// TIA Portal V20 export
FUNCTION_BLOCK "EventsPFE"   // FB95, LAD
// stored: MemoryReserve 100, Namespace Unit1.Em11, SetENOAutomatically false
   VAR
      data : Array[1..100] of LReal;
   END_VAR
BEGIN

REGION Network 1: Call PFE Events
   // Add the required PFE Events
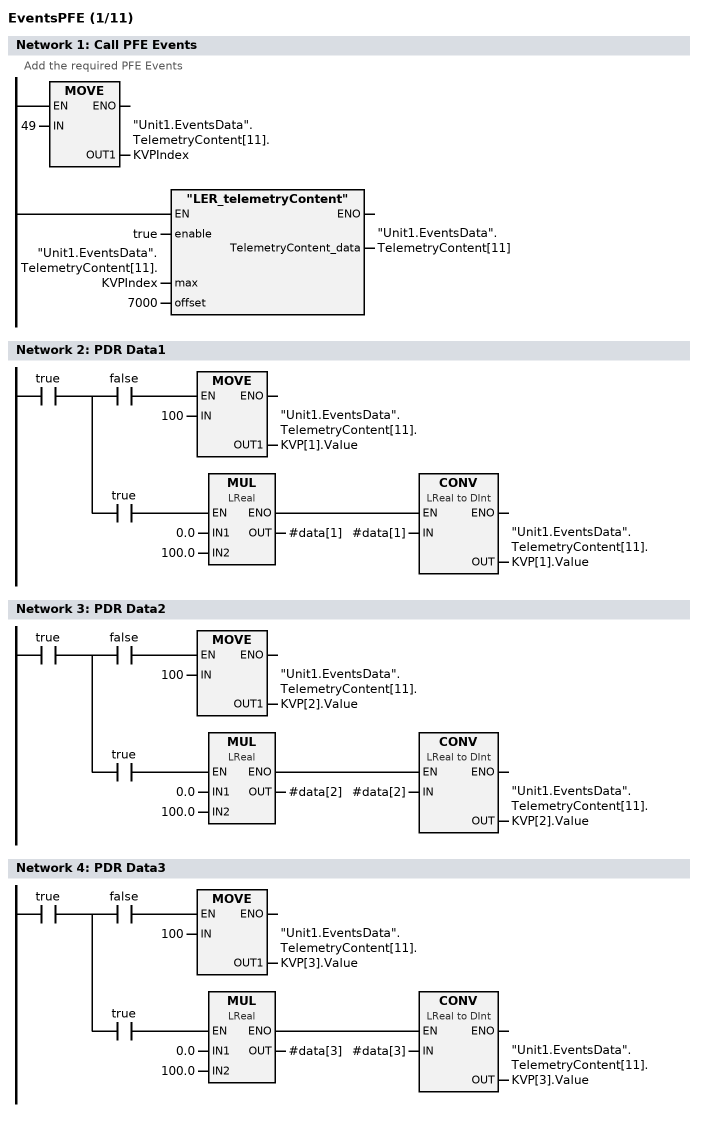
   RUNG wire#powerrail
      Move(in := 49, out1 => "Unit1.EventsData".TelemetryContent[11].KVPIndex)
   END_RUNG
   RUNG wire#powerrail
      "LER_telemetryContent"(enable := true, max := "Unit1.EventsData".TelemetryContent[11].KVPIndex, offset := 7000, TelemetryContent_data => "Unit1.EventsData".TelemetryContent[11])
   END_RUNG
   // the same network as SCL:
   "Unit1.EventsData".TelemetryContent[11].KVPIndex := 49;
   "LER_telemetryContent"(enable := true,
                          max := "Unit1.EventsData".TelemetryContent[11].KVPIndex,
                          offset := 7000,
                          TelemetryContent_data => "Unit1.EventsData".TelemetryContent[11]);
END_REGION

REGION Network 2: PDR Data1
   RUNG wire#powerrail
      Contact( true )
      wire#w1
      Contact( false )
      Move(in := 100, out1 => "Unit1.EventsData".TelemetryContent[11].KVP[1].Value)
   END_RUNG
   RUNG wire#w1
      Contact( true )
      { S7_Templates := "SrcType := LReal" } Mul(in1 := 0.0, in2 := 100.0, out => #data[1])
      { S7_Templates := "[SrcType := LReal, DestType := DInt]" } Convert(in := #data[1], out => "Unit1.EventsData".TelemetryContent[11].KVP[1].Value)
   END_RUNG
   // the same network as SCL:
   IF true AND false THEN "Unit1.EventsData".TelemetryContent[11].KVP[1].Value := 100; END_IF;
   IF true AND true THEN
       #data[1] := 0.0 * 100.0;
       "Unit1.EventsData".TelemetryContent[11].KVP[1].Value := LREAL_TO_DINT(#data[1]);
   END_IF;
END_REGION

REGION Network 3: PDR Data2
   RUNG wire#powerrail
      Contact( true )
      wire#w1
      Contact( false )
      Move(in := 100, out1 => "Unit1.EventsData".TelemetryContent[11].KVP[2].Value)
   END_RUNG
   RUNG wire#w1
      Contact( true )
      { S7_Templates := "SrcType := LReal" } Mul(in1 := 0.0, in2 := 100.0, out => #data[2])
      { S7_Templates := "[SrcType := LReal, DestType := DInt]" } Convert(in := #data[2], out => "Unit1.EventsData".TelemetryContent[11].KVP[2].Value)
   END_RUNG
   // the same network as SCL:
   IF true AND false THEN "Unit1.EventsData".TelemetryContent[11].KVP[2].Value := 100; END_IF;
   IF true AND true THEN
       #data[2] := 0.0 * 100.0;
       "Unit1.EventsData".TelemetryContent[11].KVP[2].Value := LREAL_TO_DINT(#data[2]);
   END_IF;
END_REGION

REGION Network 4: PDR Data3
   RUNG wire#powerrail
      Contact( true )
      wire#w1
      Contact( false )
      Move(in := 100, out1 => "Unit1.EventsData".TelemetryContent[11].KVP[3].Value)
   END_RUNG
   RUNG wire#w1
      Contact( true )
      { S7_Templates := "SrcType := LReal" } Mul(in1 := 0.0, in2 := 100.0, out => #data[3])
      { S7_Templates := "[SrcType := LReal, DestType := DInt]" } Convert(in := #data[3], out => "Unit1.EventsData".TelemetryContent[11].KVP[3].Value)
   END_RUNG
   // the same network as SCL:
   IF true AND false THEN "Unit1.EventsData".TelemetryContent[11].KVP[3].Value := 100; END_IF;
   IF true AND true THEN
       #data[3] := 0.0 * 100.0;
       "Unit1.EventsData".TelemetryContent[11].KVP[3].Value := LREAL_TO_DINT(#data[3]);
   END_IF;
END_REGION

REGION Network 5: PDR Data4
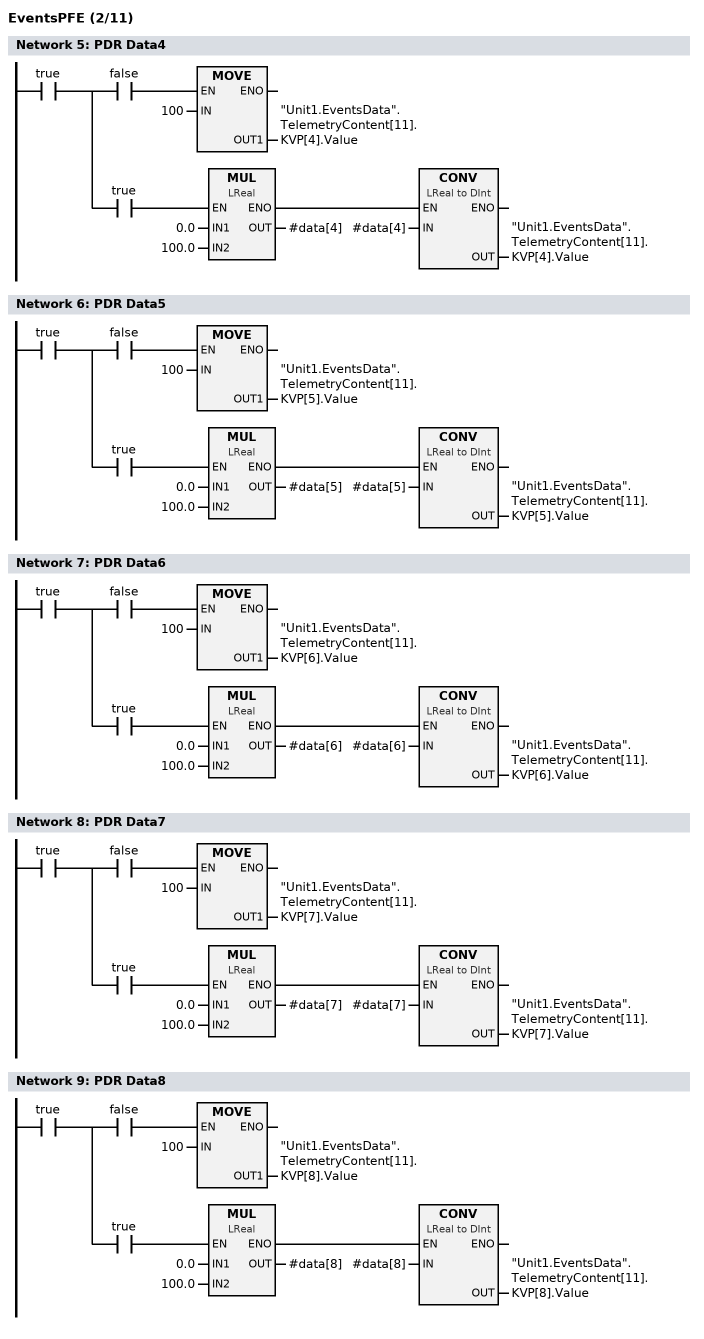
   RUNG wire#powerrail
      Contact( true )
      wire#w1
      Contact( false )
      Move(in := 100, out1 => "Unit1.EventsData".TelemetryContent[11].KVP[4].Value)
   END_RUNG
   RUNG wire#w1
      Contact( true )
      { S7_Templates := "SrcType := LReal" } Mul(in1 := 0.0, in2 := 100.0, out => #data[4])
      { S7_Templates := "[SrcType := LReal, DestType := DInt]" } Convert(in := #data[4], out => "Unit1.EventsData".TelemetryContent[11].KVP[4].Value)
   END_RUNG
   // the same network as SCL:
   IF true AND false THEN "Unit1.EventsData".TelemetryContent[11].KVP[4].Value := 100; END_IF;
   IF true AND true THEN
       #data[4] := 0.0 * 100.0;
       "Unit1.EventsData".TelemetryContent[11].KVP[4].Value := LREAL_TO_DINT(#data[4]);
   END_IF;
END_REGION

REGION Network 6: PDR Data5
   RUNG wire#powerrail
      Contact( true )
      wire#w1
      Contact( false )
      Move(in := 100, out1 => "Unit1.EventsData".TelemetryContent[11].KVP[5].Value)
   END_RUNG
   RUNG wire#w1
      Contact( true )
      { S7_Templates := "SrcType := LReal" } Mul(in1 := 0.0, in2 := 100.0, out => #data[5])
      { S7_Templates := "[SrcType := LReal, DestType := DInt]" } Convert(in := #data[5], out => "Unit1.EventsData".TelemetryContent[11].KVP[5].Value)
   END_RUNG
   // the same network as SCL:
   IF true AND false THEN "Unit1.EventsData".TelemetryContent[11].KVP[5].Value := 100; END_IF;
   IF true AND true THEN
       #data[5] := 0.0 * 100.0;
       "Unit1.EventsData".TelemetryContent[11].KVP[5].Value := LREAL_TO_DINT(#data[5]);
   END_IF;
END_REGION

REGION Network 7: PDR Data6
   RUNG wire#powerrail
      Contact( true )
      wire#w1
      Contact( false )
      Move(in := 100, out1 => "Unit1.EventsData".TelemetryContent[11].KVP[6].Value)
   END_RUNG
   RUNG wire#w1
      Contact( true )
      { S7_Templates := "SrcType := LReal" } Mul(in1 := 0.0, in2 := 100.0, out => #data[6])
      { S7_Templates := "[SrcType := LReal, DestType := DInt]" } Convert(in := #data[6], out => "Unit1.EventsData".TelemetryContent[11].KVP[6].Value)
   END_RUNG
   // the same network as SCL:
   IF true AND false THEN "Unit1.EventsData".TelemetryContent[11].KVP[6].Value := 100; END_IF;
   IF true AND true THEN
       #data[6] := 0.0 * 100.0;
       "Unit1.EventsData".TelemetryContent[11].KVP[6].Value := LREAL_TO_DINT(#data[6]);
   END_IF;
END_REGION

REGION Network 8: PDR Data7
   RUNG wire#powerrail
      Contact( true )
      wire#w1
      Contact( false )
      Move(in := 100, out1 => "Unit1.EventsData".TelemetryContent[11].KVP[7].Value)
   END_RUNG
   RUNG wire#w1
      Contact( true )
      { S7_Templates := "SrcType := LReal" } Mul(in1 := 0.0, in2 := 100.0, out => #data[7])
      { S7_Templates := "[SrcType := LReal, DestType := DInt]" } Convert(in := #data[7], out => "Unit1.EventsData".TelemetryContent[11].KVP[7].Value)
   END_RUNG
   // the same network as SCL:
   IF true AND false THEN "Unit1.EventsData".TelemetryContent[11].KVP[7].Value := 100; END_IF;
   IF true AND true THEN
       #data[7] := 0.0 * 100.0;
       "Unit1.EventsData".TelemetryContent[11].KVP[7].Value := LREAL_TO_DINT(#data[7]);
   END_IF;
END_REGION

REGION Network 9: PDR Data8
   RUNG wire#powerrail
      Contact( true )
      wire#w1
      Contact( false )
      Move(in := 100, out1 => "Unit1.EventsData".TelemetryContent[11].KVP[8].Value)
   END_RUNG
   RUNG wire#w1
      Contact( true )
      { S7_Templates := "SrcType := LReal" } Mul(in1 := 0.0, in2 := 100.0, out => #data[8])
      { S7_Templates := "[SrcType := LReal, DestType := DInt]" } Convert(in := #data[8], out => "Unit1.EventsData".TelemetryContent[11].KVP[8].Value)
   END_RUNG
   // the same network as SCL:
   IF true AND false THEN "Unit1.EventsData".TelemetryContent[11].KVP[8].Value := 100; END_IF;
   IF true AND true THEN
       #data[8] := 0.0 * 100.0;
       "Unit1.EventsData".TelemetryContent[11].KVP[8].Value := LREAL_TO_DINT(#data[8]);
   END_IF;
END_REGION

REGION Network 10: PDR Data9
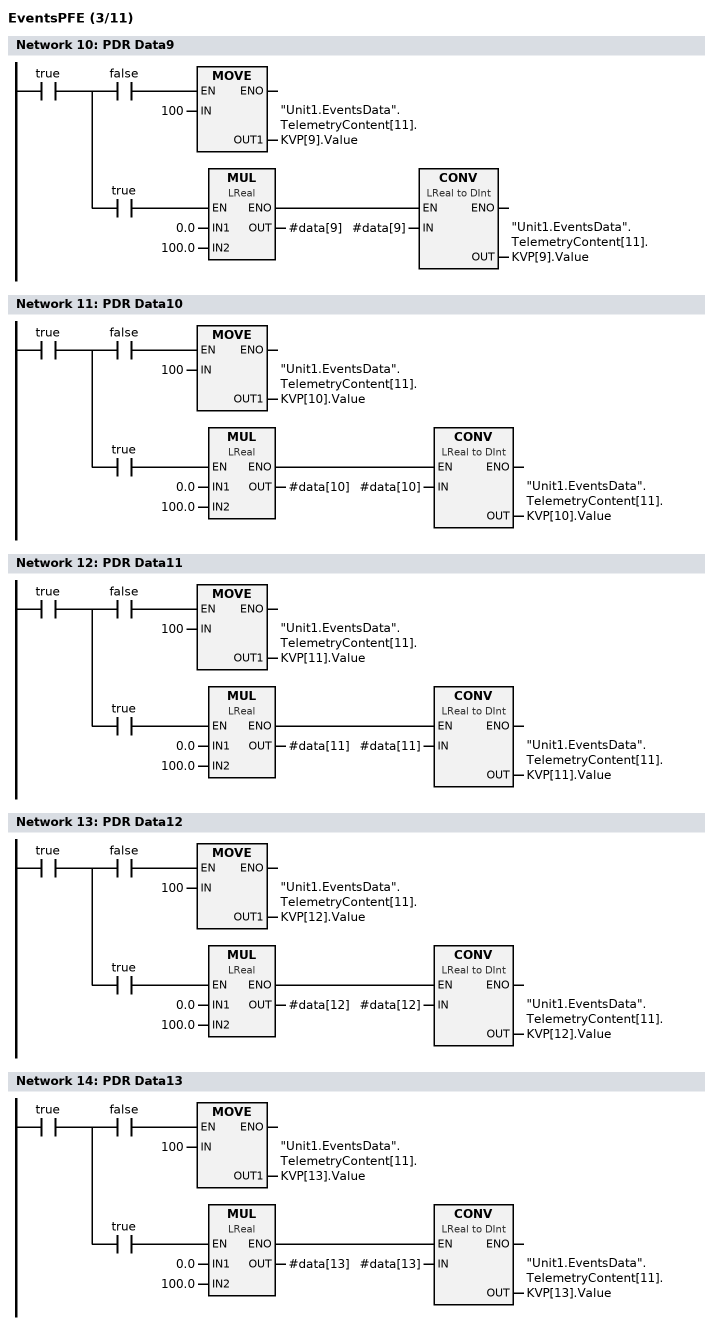
   RUNG wire#powerrail
      Contact( true )
      wire#w1
      Contact( false )
      Move(in := 100, out1 => "Unit1.EventsData".TelemetryContent[11].KVP[9].Value)
   END_RUNG
   RUNG wire#w1
      Contact( true )
      { S7_Templates := "SrcType := LReal" } Mul(in1 := 0.0, in2 := 100.0, out => #data[9])
      { S7_Templates := "[SrcType := LReal, DestType := DInt]" } Convert(in := #data[9], out => "Unit1.EventsData".TelemetryContent[11].KVP[9].Value)
   END_RUNG
   // the same network as SCL:
   IF true AND false THEN "Unit1.EventsData".TelemetryContent[11].KVP[9].Value := 100; END_IF;
   IF true AND true THEN
       #data[9] := 0.0 * 100.0;
       "Unit1.EventsData".TelemetryContent[11].KVP[9].Value := LREAL_TO_DINT(#data[9]);
   END_IF;
END_REGION

REGION Network 11: PDR Data10
   RUNG wire#powerrail
      Contact( true )
      wire#w1
      Contact( false )
      Move(in := 100, out1 => "Unit1.EventsData".TelemetryContent[11].KVP[10].Value)
   END_RUNG
   RUNG wire#w1
      Contact( true )
      { S7_Templates := "SrcType := LReal" } Mul(in1 := 0.0, in2 := 100.0, out => #data[10])
      { S7_Templates := "[SrcType := LReal, DestType := DInt]" } Convert(in := #data[10], out => "Unit1.EventsData".TelemetryContent[11].KVP[10].Value)
   END_RUNG
   // the same network as SCL:
   IF true AND false THEN "Unit1.EventsData".TelemetryContent[11].KVP[10].Value := 100; END_IF;
   IF true AND true THEN
       #data[10] := 0.0 * 100.0;
       "Unit1.EventsData".TelemetryContent[11].KVP[10].Value := LREAL_TO_DINT(#data[10]);
   END_IF;
END_REGION

REGION Network 12: PDR Data11
   RUNG wire#powerrail
      Contact( true )
      wire#w1
      Contact( false )
      Move(in := 100, out1 => "Unit1.EventsData".TelemetryContent[11].KVP[11].Value)
   END_RUNG
   RUNG wire#w1
      Contact( true )
      { S7_Templates := "SrcType := LReal" } Mul(in1 := 0.0, in2 := 100.0, out => #data[11])
      { S7_Templates := "[SrcType := LReal, DestType := DInt]" } Convert(in := #data[11], out => "Unit1.EventsData".TelemetryContent[11].KVP[11].Value)
   END_RUNG
   // the same network as SCL:
   IF true AND false THEN "Unit1.EventsData".TelemetryContent[11].KVP[11].Value := 100; END_IF;
   IF true AND true THEN
       #data[11] := 0.0 * 100.0;
       "Unit1.EventsData".TelemetryContent[11].KVP[11].Value := LREAL_TO_DINT(#data[11]);
   END_IF;
END_REGION

REGION Network 13: PDR Data12
   RUNG wire#powerrail
      Contact( true )
      wire#w1
      Contact( false )
      Move(in := 100, out1 => "Unit1.EventsData".TelemetryContent[11].KVP[12].Value)
   END_RUNG
   RUNG wire#w1
      Contact( true )
      { S7_Templates := "SrcType := LReal" } Mul(in1 := 0.0, in2 := 100.0, out => #data[12])
      { S7_Templates := "[SrcType := LReal, DestType := DInt]" } Convert(in := #data[12], out => "Unit1.EventsData".TelemetryContent[11].KVP[12].Value)
   END_RUNG
   // the same network as SCL:
   IF true AND false THEN "Unit1.EventsData".TelemetryContent[11].KVP[12].Value := 100; END_IF;
   IF true AND true THEN
       #data[12] := 0.0 * 100.0;
       "Unit1.EventsData".TelemetryContent[11].KVP[12].Value := LREAL_TO_DINT(#data[12]);
   END_IF;
END_REGION

REGION Network 14: PDR Data13
   RUNG wire#powerrail
      Contact( true )
      wire#w1
      Contact( false )
      Move(in := 100, out1 => "Unit1.EventsData".TelemetryContent[11].KVP[13].Value)
   END_RUNG
   RUNG wire#w1
      Contact( true )
      { S7_Templates := "SrcType := LReal" } Mul(in1 := 0.0, in2 := 100.0, out => #data[13])
      { S7_Templates := "[SrcType := LReal, DestType := DInt]" } Convert(in := #data[13], out => "Unit1.EventsData".TelemetryContent[11].KVP[13].Value)
   END_RUNG
   // the same network as SCL:
   IF true AND false THEN "Unit1.EventsData".TelemetryContent[11].KVP[13].Value := 100; END_IF;
   IF true AND true THEN
       #data[13] := 0.0 * 100.0;
       "Unit1.EventsData".TelemetryContent[11].KVP[13].Value := LREAL_TO_DINT(#data[13]);
   END_IF;
END_REGION

REGION Network 15: PDR Data14
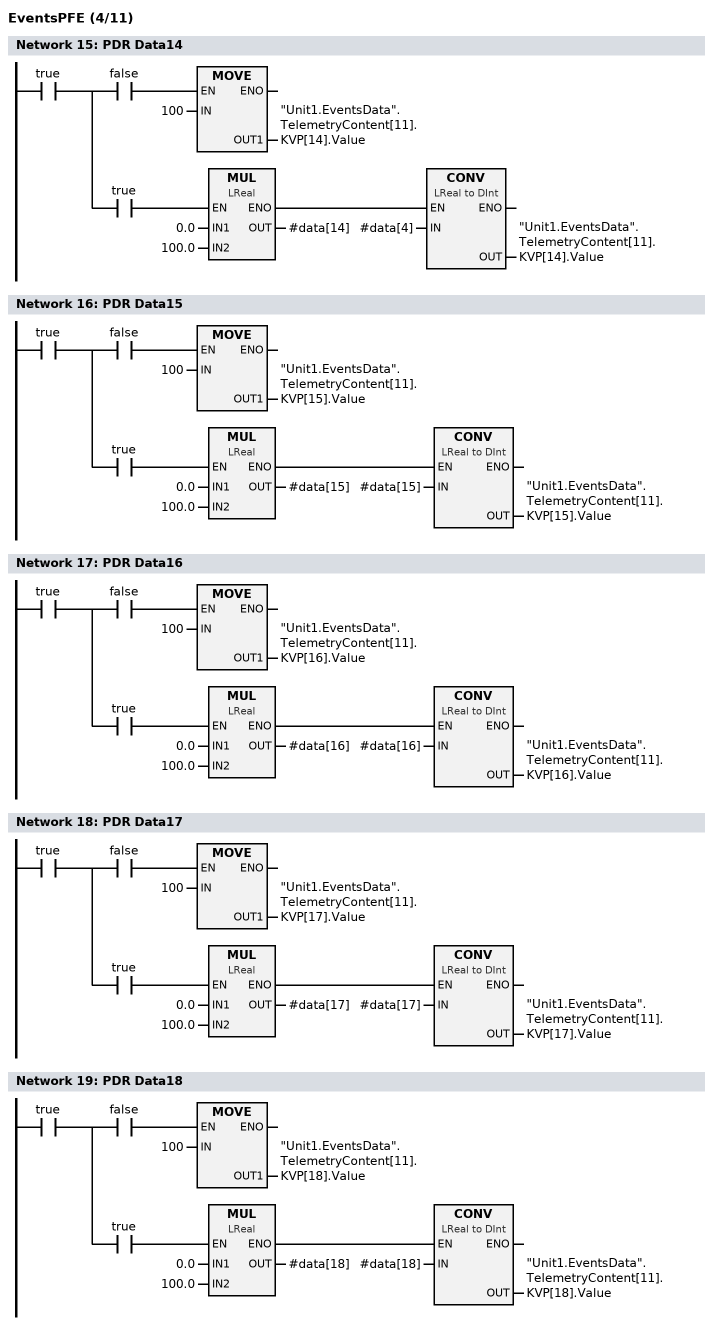
   RUNG wire#powerrail
      Contact( true )
      wire#w1
      Contact( false )
      Move(in := 100, out1 => "Unit1.EventsData".TelemetryContent[11].KVP[14].Value)
   END_RUNG
   RUNG wire#w1
      Contact( true )
      { S7_Templates := "SrcType := LReal" } Mul(in1 := 0.0, in2 := 100.0, out => #data[14])
      { S7_Templates := "[SrcType := LReal, DestType := DInt]" } Convert(in := #data[4], out => "Unit1.EventsData".TelemetryContent[11].KVP[14].Value)
   END_RUNG
   // the same network as SCL:
   IF true AND false THEN "Unit1.EventsData".TelemetryContent[11].KVP[14].Value := 100; END_IF;
   IF true AND true THEN
       #data[14] := 0.0 * 100.0;
       "Unit1.EventsData".TelemetryContent[11].KVP[14].Value := LREAL_TO_DINT(#data[4]);
   END_IF;
END_REGION

REGION Network 16: PDR Data15
   RUNG wire#powerrail
      Contact( true )
      wire#w1
      Contact( false )
      Move(in := 100, out1 => "Unit1.EventsData".TelemetryContent[11].KVP[15].Value)
   END_RUNG
   RUNG wire#w1
      Contact( true )
      { S7_Templates := "SrcType := LReal" } Mul(in1 := 0.0, in2 := 100.0, out => #data[15])
      { S7_Templates := "[SrcType := LReal, DestType := DInt]" } Convert(in := #data[15], out => "Unit1.EventsData".TelemetryContent[11].KVP[15].Value)
   END_RUNG
   // the same network as SCL:
   IF true AND false THEN "Unit1.EventsData".TelemetryContent[11].KVP[15].Value := 100; END_IF;
   IF true AND true THEN
       #data[15] := 0.0 * 100.0;
       "Unit1.EventsData".TelemetryContent[11].KVP[15].Value := LREAL_TO_DINT(#data[15]);
   END_IF;
END_REGION

REGION Network 17: PDR Data16
   RUNG wire#powerrail
      Contact( true )
      wire#w1
      Contact( false )
      Move(in := 100, out1 => "Unit1.EventsData".TelemetryContent[11].KVP[16].Value)
   END_RUNG
   RUNG wire#w1
      Contact( true )
      { S7_Templates := "SrcType := LReal" } Mul(in1 := 0.0, in2 := 100.0, out => #data[16])
      { S7_Templates := "[SrcType := LReal, DestType := DInt]" } Convert(in := #data[16], out => "Unit1.EventsData".TelemetryContent[11].KVP[16].Value)
   END_RUNG
   // the same network as SCL:
   IF true AND false THEN "Unit1.EventsData".TelemetryContent[11].KVP[16].Value := 100; END_IF;
   IF true AND true THEN
       #data[16] := 0.0 * 100.0;
       "Unit1.EventsData".TelemetryContent[11].KVP[16].Value := LREAL_TO_DINT(#data[16]);
   END_IF;
END_REGION

REGION Network 18: PDR Data17
   RUNG wire#powerrail
      Contact( true )
      wire#w1
      Contact( false )
      Move(in := 100, out1 => "Unit1.EventsData".TelemetryContent[11].KVP[17].Value)
   END_RUNG
   RUNG wire#w1
      Contact( true )
      { S7_Templates := "SrcType := LReal" } Mul(in1 := 0.0, in2 := 100.0, out => #data[17])
      { S7_Templates := "[SrcType := LReal, DestType := DInt]" } Convert(in := #data[17], out => "Unit1.EventsData".TelemetryContent[11].KVP[17].Value)
   END_RUNG
   // the same network as SCL:
   IF true AND false THEN "Unit1.EventsData".TelemetryContent[11].KVP[17].Value := 100; END_IF;
   IF true AND true THEN
       #data[17] := 0.0 * 100.0;
       "Unit1.EventsData".TelemetryContent[11].KVP[17].Value := LREAL_TO_DINT(#data[17]);
   END_IF;
END_REGION

REGION Network 19: PDR Data18
   RUNG wire#powerrail
      Contact( true )
      wire#w1
      Contact( false )
      Move(in := 100, out1 => "Unit1.EventsData".TelemetryContent[11].KVP[18].Value)
   END_RUNG
   RUNG wire#w1
      Contact( true )
      { S7_Templates := "SrcType := LReal" } Mul(in1 := 0.0, in2 := 100.0, out => #data[18])
      { S7_Templates := "[SrcType := LReal, DestType := DInt]" } Convert(in := #data[18], out => "Unit1.EventsData".TelemetryContent[11].KVP[18].Value)
   END_RUNG
   // the same network as SCL:
   IF true AND false THEN "Unit1.EventsData".TelemetryContent[11].KVP[18].Value := 100; END_IF;
   IF true AND true THEN
       #data[18] := 0.0 * 100.0;
       "Unit1.EventsData".TelemetryContent[11].KVP[18].Value := LREAL_TO_DINT(#data[18]);
   END_IF;
END_REGION

REGION Network 20: PDR Data19
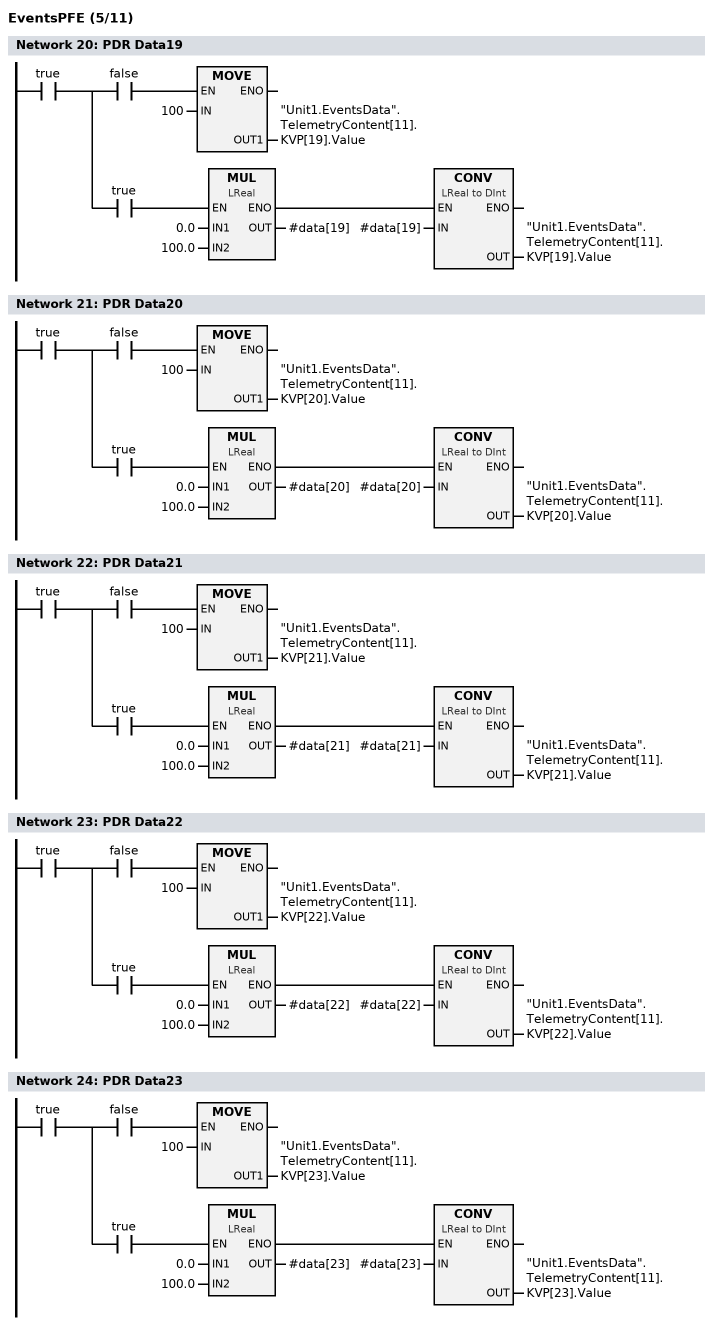
   RUNG wire#powerrail
      Contact( true )
      wire#w1
      Contact( false )
      Move(in := 100, out1 => "Unit1.EventsData".TelemetryContent[11].KVP[19].Value)
   END_RUNG
   RUNG wire#w1
      Contact( true )
      { S7_Templates := "SrcType := LReal" } Mul(in1 := 0.0, in2 := 100.0, out => #data[19])
      { S7_Templates := "[SrcType := LReal, DestType := DInt]" } Convert(in := #data[19], out => "Unit1.EventsData".TelemetryContent[11].KVP[19].Value)
   END_RUNG
   // the same network as SCL:
   IF true AND false THEN "Unit1.EventsData".TelemetryContent[11].KVP[19].Value := 100; END_IF;
   IF true AND true THEN
       #data[19] := 0.0 * 100.0;
       "Unit1.EventsData".TelemetryContent[11].KVP[19].Value := LREAL_TO_DINT(#data[19]);
   END_IF;
END_REGION

REGION Network 21: PDR Data20
   RUNG wire#powerrail
      Contact( true )
      wire#w1
      Contact( false )
      Move(in := 100, out1 => "Unit1.EventsData".TelemetryContent[11].KVP[20].Value)
   END_RUNG
   RUNG wire#w1
      Contact( true )
      { S7_Templates := "SrcType := LReal" } Mul(in1 := 0.0, in2 := 100.0, out => #data[20])
      { S7_Templates := "[SrcType := LReal, DestType := DInt]" } Convert(in := #data[20], out => "Unit1.EventsData".TelemetryContent[11].KVP[20].Value)
   END_RUNG
   // the same network as SCL:
   IF true AND false THEN "Unit1.EventsData".TelemetryContent[11].KVP[20].Value := 100; END_IF;
   IF true AND true THEN
       #data[20] := 0.0 * 100.0;
       "Unit1.EventsData".TelemetryContent[11].KVP[20].Value := LREAL_TO_DINT(#data[20]);
   END_IF;
END_REGION

REGION Network 22: PDR Data21
   RUNG wire#powerrail
      Contact( true )
      wire#w1
      Contact( false )
      Move(in := 100, out1 => "Unit1.EventsData".TelemetryContent[11].KVP[21].Value)
   END_RUNG
   RUNG wire#w1
      Contact( true )
      { S7_Templates := "SrcType := LReal" } Mul(in1 := 0.0, in2 := 100.0, out => #data[21])
      { S7_Templates := "[SrcType := LReal, DestType := DInt]" } Convert(in := #data[21], out => "Unit1.EventsData".TelemetryContent[11].KVP[21].Value)
   END_RUNG
   // the same network as SCL:
   IF true AND false THEN "Unit1.EventsData".TelemetryContent[11].KVP[21].Value := 100; END_IF;
   IF true AND true THEN
       #data[21] := 0.0 * 100.0;
       "Unit1.EventsData".TelemetryContent[11].KVP[21].Value := LREAL_TO_DINT(#data[21]);
   END_IF;
END_REGION

REGION Network 23: PDR Data22
   RUNG wire#powerrail
      Contact( true )
      wire#w1
      Contact( false )
      Move(in := 100, out1 => "Unit1.EventsData".TelemetryContent[11].KVP[22].Value)
   END_RUNG
   RUNG wire#w1
      Contact( true )
      { S7_Templates := "SrcType := LReal" } Mul(in1 := 0.0, in2 := 100.0, out => #data[22])
      { S7_Templates := "[SrcType := LReal, DestType := DInt]" } Convert(in := #data[22], out => "Unit1.EventsData".TelemetryContent[11].KVP[22].Value)
   END_RUNG
   // the same network as SCL:
   IF true AND false THEN "Unit1.EventsData".TelemetryContent[11].KVP[22].Value := 100; END_IF;
   IF true AND true THEN
       #data[22] := 0.0 * 100.0;
       "Unit1.EventsData".TelemetryContent[11].KVP[22].Value := LREAL_TO_DINT(#data[22]);
   END_IF;
END_REGION

REGION Network 24: PDR Data23
   RUNG wire#powerrail
      Contact( true )
      wire#w1
      Contact( false )
      Move(in := 100, out1 => "Unit1.EventsData".TelemetryContent[11].KVP[23].Value)
   END_RUNG
   RUNG wire#w1
      Contact( true )
      { S7_Templates := "SrcType := LReal" } Mul(in1 := 0.0, in2 := 100.0, out => #data[23])
      { S7_Templates := "[SrcType := LReal, DestType := DInt]" } Convert(in := #data[23], out => "Unit1.EventsData".TelemetryContent[11].KVP[23].Value)
   END_RUNG
   // the same network as SCL:
   IF true AND false THEN "Unit1.EventsData".TelemetryContent[11].KVP[23].Value := 100; END_IF;
   IF true AND true THEN
       #data[23] := 0.0 * 100.0;
       "Unit1.EventsData".TelemetryContent[11].KVP[23].Value := LREAL_TO_DINT(#data[23]);
   END_IF;
END_REGION

REGION Network 25: PDR Data24
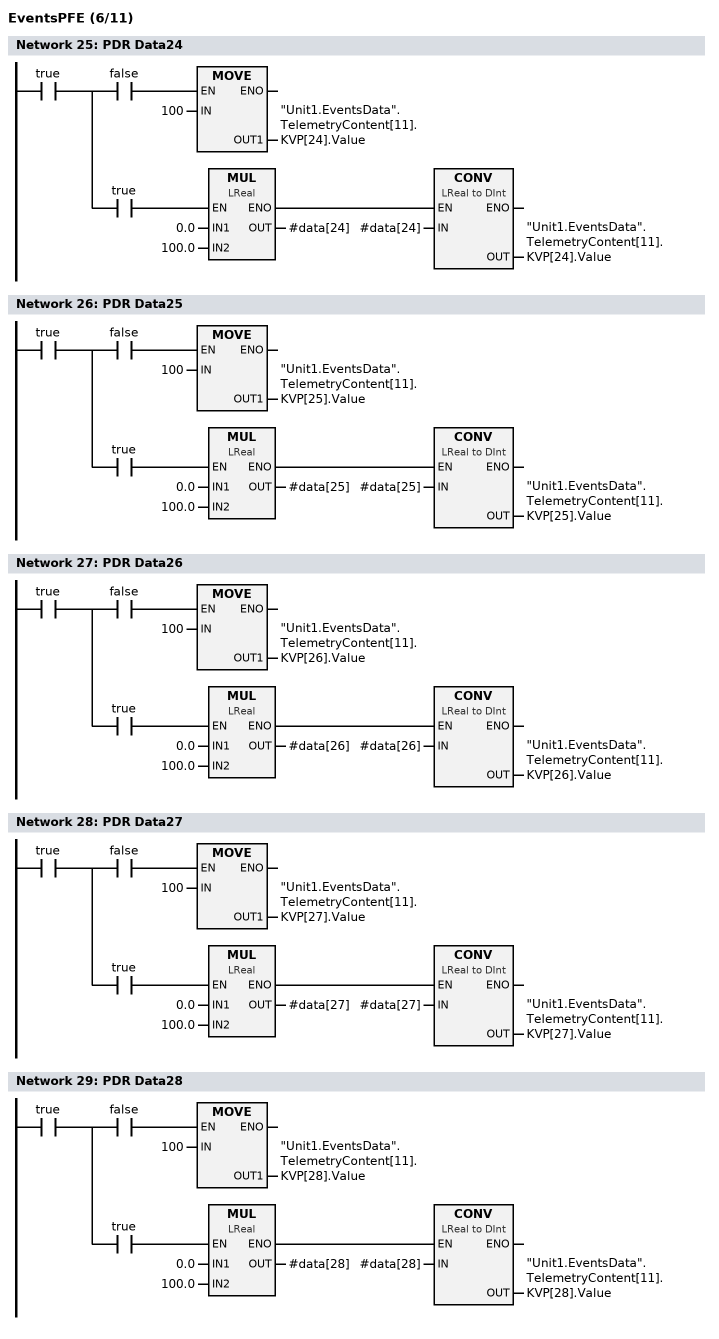
   RUNG wire#powerrail
      Contact( true )
      wire#w1
      Contact( false )
      Move(in := 100, out1 => "Unit1.EventsData".TelemetryContent[11].KVP[24].Value)
   END_RUNG
   RUNG wire#w1
      Contact( true )
      { S7_Templates := "SrcType := LReal" } Mul(in1 := 0.0, in2 := 100.0, out => #data[24])
      { S7_Templates := "[SrcType := LReal, DestType := DInt]" } Convert(in := #data[24], out => "Unit1.EventsData".TelemetryContent[11].KVP[24].Value)
   END_RUNG
   // the same network as SCL:
   IF true AND false THEN "Unit1.EventsData".TelemetryContent[11].KVP[24].Value := 100; END_IF;
   IF true AND true THEN
       #data[24] := 0.0 * 100.0;
       "Unit1.EventsData".TelemetryContent[11].KVP[24].Value := LREAL_TO_DINT(#data[24]);
   END_IF;
END_REGION

REGION Network 26: PDR Data25
   RUNG wire#powerrail
      Contact( true )
      wire#w1
      Contact( false )
      Move(in := 100, out1 => "Unit1.EventsData".TelemetryContent[11].KVP[25].Value)
   END_RUNG
   RUNG wire#w1
      Contact( true )
      { S7_Templates := "SrcType := LReal" } Mul(in1 := 0.0, in2 := 100.0, out => #data[25])
      { S7_Templates := "[SrcType := LReal, DestType := DInt]" } Convert(in := #data[25], out => "Unit1.EventsData".TelemetryContent[11].KVP[25].Value)
   END_RUNG
   // the same network as SCL:
   IF true AND false THEN "Unit1.EventsData".TelemetryContent[11].KVP[25].Value := 100; END_IF;
   IF true AND true THEN
       #data[25] := 0.0 * 100.0;
       "Unit1.EventsData".TelemetryContent[11].KVP[25].Value := LREAL_TO_DINT(#data[25]);
   END_IF;
END_REGION

REGION Network 27: PDR Data26
   RUNG wire#powerrail
      Contact( true )
      wire#w1
      Contact( false )
      Move(in := 100, out1 => "Unit1.EventsData".TelemetryContent[11].KVP[26].Value)
   END_RUNG
   RUNG wire#w1
      Contact( true )
      { S7_Templates := "SrcType := LReal" } Mul(in1 := 0.0, in2 := 100.0, out => #data[26])
      { S7_Templates := "[SrcType := LReal, DestType := DInt]" } Convert(in := #data[26], out => "Unit1.EventsData".TelemetryContent[11].KVP[26].Value)
   END_RUNG
   // the same network as SCL:
   IF true AND false THEN "Unit1.EventsData".TelemetryContent[11].KVP[26].Value := 100; END_IF;
   IF true AND true THEN
       #data[26] := 0.0 * 100.0;
       "Unit1.EventsData".TelemetryContent[11].KVP[26].Value := LREAL_TO_DINT(#data[26]);
   END_IF;
END_REGION

REGION Network 28: PDR Data27
   RUNG wire#powerrail
      Contact( true )
      wire#w1
      Contact( false )
      Move(in := 100, out1 => "Unit1.EventsData".TelemetryContent[11].KVP[27].Value)
   END_RUNG
   RUNG wire#w1
      Contact( true )
      { S7_Templates := "SrcType := LReal" } Mul(in1 := 0.0, in2 := 100.0, out => #data[27])
      { S7_Templates := "[SrcType := LReal, DestType := DInt]" } Convert(in := #data[27], out => "Unit1.EventsData".TelemetryContent[11].KVP[27].Value)
   END_RUNG
   // the same network as SCL:
   IF true AND false THEN "Unit1.EventsData".TelemetryContent[11].KVP[27].Value := 100; END_IF;
   IF true AND true THEN
       #data[27] := 0.0 * 100.0;
       "Unit1.EventsData".TelemetryContent[11].KVP[27].Value := LREAL_TO_DINT(#data[27]);
   END_IF;
END_REGION

REGION Network 29: PDR Data28
   RUNG wire#powerrail
      Contact( true )
      wire#w1
      Contact( false )
      Move(in := 100, out1 => "Unit1.EventsData".TelemetryContent[11].KVP[28].Value)
   END_RUNG
   RUNG wire#w1
      Contact( true )
      { S7_Templates := "SrcType := LReal" } Mul(in1 := 0.0, in2 := 100.0, out => #data[28])
      { S7_Templates := "[SrcType := LReal, DestType := DInt]" } Convert(in := #data[28], out => "Unit1.EventsData".TelemetryContent[11].KVP[28].Value)
   END_RUNG
   // the same network as SCL:
   IF true AND false THEN "Unit1.EventsData".TelemetryContent[11].KVP[28].Value := 100; END_IF;
   IF true AND true THEN
       #data[28] := 0.0 * 100.0;
       "Unit1.EventsData".TelemetryContent[11].KVP[28].Value := LREAL_TO_DINT(#data[28]);
   END_IF;
END_REGION

REGION Network 30: PDR Data29
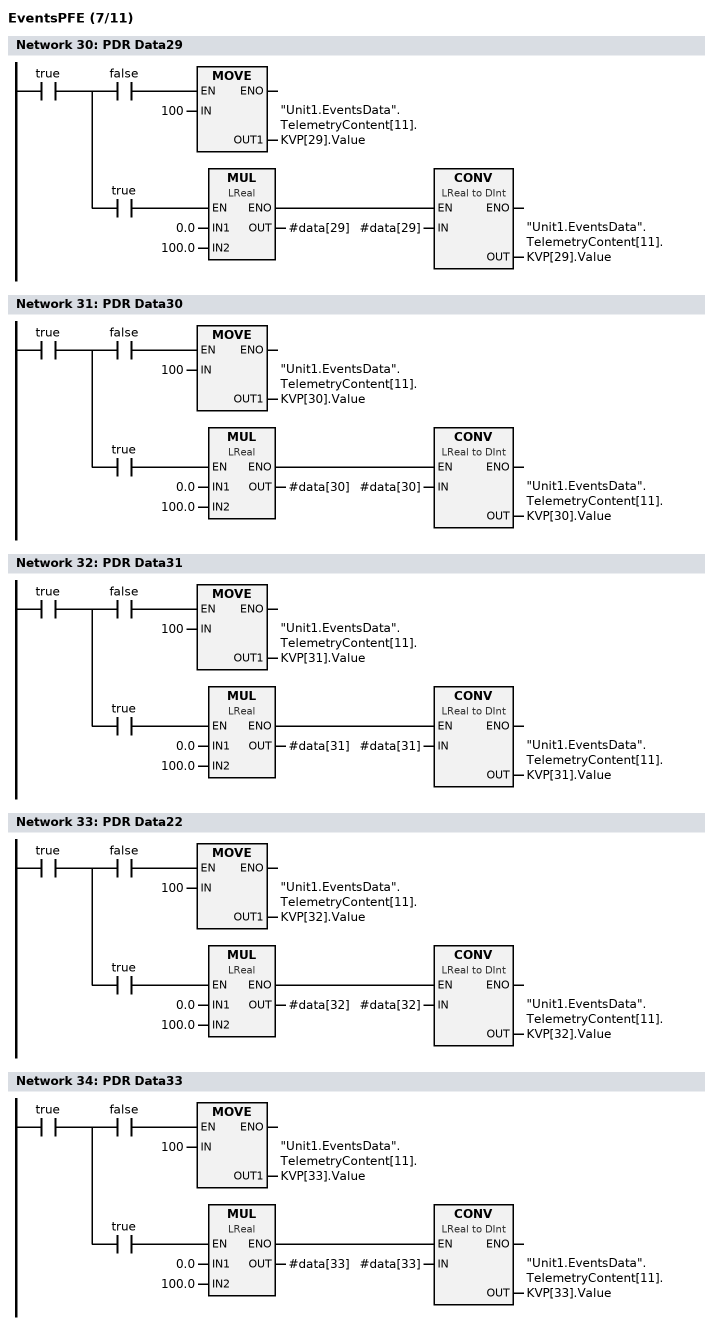
   RUNG wire#powerrail
      Contact( true )
      wire#w1
      Contact( false )
      Move(in := 100, out1 => "Unit1.EventsData".TelemetryContent[11].KVP[29].Value)
   END_RUNG
   RUNG wire#w1
      Contact( true )
      { S7_Templates := "SrcType := LReal" } Mul(in1 := 0.0, in2 := 100.0, out => #data[29])
      { S7_Templates := "[SrcType := LReal, DestType := DInt]" } Convert(in := #data[29], out => "Unit1.EventsData".TelemetryContent[11].KVP[29].Value)
   END_RUNG
   // the same network as SCL:
   IF true AND false THEN "Unit1.EventsData".TelemetryContent[11].KVP[29].Value := 100; END_IF;
   IF true AND true THEN
       #data[29] := 0.0 * 100.0;
       "Unit1.EventsData".TelemetryContent[11].KVP[29].Value := LREAL_TO_DINT(#data[29]);
   END_IF;
END_REGION

REGION Network 31: PDR Data30
   RUNG wire#powerrail
      Contact( true )
      wire#w1
      Contact( false )
      Move(in := 100, out1 => "Unit1.EventsData".TelemetryContent[11].KVP[30].Value)
   END_RUNG
   RUNG wire#w1
      Contact( true )
      { S7_Templates := "SrcType := LReal" } Mul(in1 := 0.0, in2 := 100.0, out => #data[30])
      { S7_Templates := "[SrcType := LReal, DestType := DInt]" } Convert(in := #data[30], out => "Unit1.EventsData".TelemetryContent[11].KVP[30].Value)
   END_RUNG
   // the same network as SCL:
   IF true AND false THEN "Unit1.EventsData".TelemetryContent[11].KVP[30].Value := 100; END_IF;
   IF true AND true THEN
       #data[30] := 0.0 * 100.0;
       "Unit1.EventsData".TelemetryContent[11].KVP[30].Value := LREAL_TO_DINT(#data[30]);
   END_IF;
END_REGION

REGION Network 32: PDR Data31
   RUNG wire#powerrail
      Contact( true )
      wire#w1
      Contact( false )
      Move(in := 100, out1 => "Unit1.EventsData".TelemetryContent[11].KVP[31].Value)
   END_RUNG
   RUNG wire#w1
      Contact( true )
      { S7_Templates := "SrcType := LReal" } Mul(in1 := 0.0, in2 := 100.0, out => #data[31])
      { S7_Templates := "[SrcType := LReal, DestType := DInt]" } Convert(in := #data[31], out => "Unit1.EventsData".TelemetryContent[11].KVP[31].Value)
   END_RUNG
   // the same network as SCL:
   IF true AND false THEN "Unit1.EventsData".TelemetryContent[11].KVP[31].Value := 100; END_IF;
   IF true AND true THEN
       #data[31] := 0.0 * 100.0;
       "Unit1.EventsData".TelemetryContent[11].KVP[31].Value := LREAL_TO_DINT(#data[31]);
   END_IF;
END_REGION

REGION Network 33: PDR Data22
   RUNG wire#powerrail
      Contact( true )
      wire#w1
      Contact( false )
      Move(in := 100, out1 => "Unit1.EventsData".TelemetryContent[11].KVP[32].Value)
   END_RUNG
   RUNG wire#w1
      Contact( true )
      { S7_Templates := "SrcType := LReal" } Mul(in1 := 0.0, in2 := 100.0, out => #data[32])
      { S7_Templates := "[SrcType := LReal, DestType := DInt]" } Convert(in := #data[32], out => "Unit1.EventsData".TelemetryContent[11].KVP[32].Value)
   END_RUNG
   // the same network as SCL:
   IF true AND false THEN "Unit1.EventsData".TelemetryContent[11].KVP[32].Value := 100; END_IF;
   IF true AND true THEN
       #data[32] := 0.0 * 100.0;
       "Unit1.EventsData".TelemetryContent[11].KVP[32].Value := LREAL_TO_DINT(#data[32]);
   END_IF;
END_REGION

REGION Network 34: PDR Data33
   RUNG wire#powerrail
      Contact( true )
      wire#w1
      Contact( false )
      Move(in := 100, out1 => "Unit1.EventsData".TelemetryContent[11].KVP[33].Value)
   END_RUNG
   RUNG wire#w1
      Contact( true )
      { S7_Templates := "SrcType := LReal" } Mul(in1 := 0.0, in2 := 100.0, out => #data[33])
      { S7_Templates := "[SrcType := LReal, DestType := DInt]" } Convert(in := #data[33], out => "Unit1.EventsData".TelemetryContent[11].KVP[33].Value)
   END_RUNG
   // the same network as SCL:
   IF true AND false THEN "Unit1.EventsData".TelemetryContent[11].KVP[33].Value := 100; END_IF;
   IF true AND true THEN
       #data[33] := 0.0 * 100.0;
       "Unit1.EventsData".TelemetryContent[11].KVP[33].Value := LREAL_TO_DINT(#data[33]);
   END_IF;
END_REGION

REGION Network 35: PDR Data34
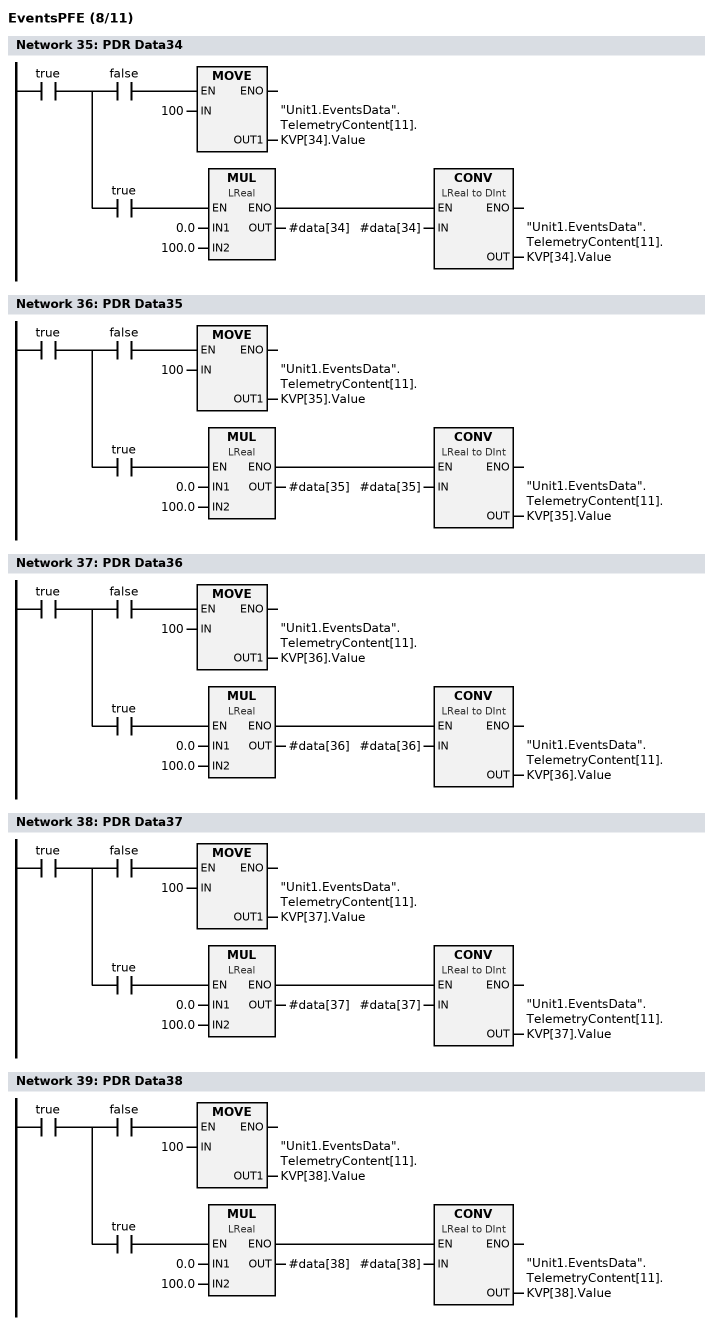
   RUNG wire#powerrail
      Contact( true )
      wire#w1
      Contact( false )
      Move(in := 100, out1 => "Unit1.EventsData".TelemetryContent[11].KVP[34].Value)
   END_RUNG
   RUNG wire#w1
      Contact( true )
      { S7_Templates := "SrcType := LReal" } Mul(in1 := 0.0, in2 := 100.0, out => #data[34])
      { S7_Templates := "[SrcType := LReal, DestType := DInt]" } Convert(in := #data[34], out => "Unit1.EventsData".TelemetryContent[11].KVP[34].Value)
   END_RUNG
   // the same network as SCL:
   IF true AND false THEN "Unit1.EventsData".TelemetryContent[11].KVP[34].Value := 100; END_IF;
   IF true AND true THEN
       #data[34] := 0.0 * 100.0;
       "Unit1.EventsData".TelemetryContent[11].KVP[34].Value := LREAL_TO_DINT(#data[34]);
   END_IF;
END_REGION

REGION Network 36: PDR Data35
   RUNG wire#powerrail
      Contact( true )
      wire#w1
      Contact( false )
      Move(in := 100, out1 => "Unit1.EventsData".TelemetryContent[11].KVP[35].Value)
   END_RUNG
   RUNG wire#w1
      Contact( true )
      { S7_Templates := "SrcType := LReal" } Mul(in1 := 0.0, in2 := 100.0, out => #data[35])
      { S7_Templates := "[SrcType := LReal, DestType := DInt]" } Convert(in := #data[35], out => "Unit1.EventsData".TelemetryContent[11].KVP[35].Value)
   END_RUNG
   // the same network as SCL:
   IF true AND false THEN "Unit1.EventsData".TelemetryContent[11].KVP[35].Value := 100; END_IF;
   IF true AND true THEN
       #data[35] := 0.0 * 100.0;
       "Unit1.EventsData".TelemetryContent[11].KVP[35].Value := LREAL_TO_DINT(#data[35]);
   END_IF;
END_REGION

REGION Network 37: PDR Data36
   RUNG wire#powerrail
      Contact( true )
      wire#w1
      Contact( false )
      Move(in := 100, out1 => "Unit1.EventsData".TelemetryContent[11].KVP[36].Value)
   END_RUNG
   RUNG wire#w1
      Contact( true )
      { S7_Templates := "SrcType := LReal" } Mul(in1 := 0.0, in2 := 100.0, out => #data[36])
      { S7_Templates := "[SrcType := LReal, DestType := DInt]" } Convert(in := #data[36], out => "Unit1.EventsData".TelemetryContent[11].KVP[36].Value)
   END_RUNG
   // the same network as SCL:
   IF true AND false THEN "Unit1.EventsData".TelemetryContent[11].KVP[36].Value := 100; END_IF;
   IF true AND true THEN
       #data[36] := 0.0 * 100.0;
       "Unit1.EventsData".TelemetryContent[11].KVP[36].Value := LREAL_TO_DINT(#data[36]);
   END_IF;
END_REGION

REGION Network 38: PDR Data37
   RUNG wire#powerrail
      Contact( true )
      wire#w1
      Contact( false )
      Move(in := 100, out1 => "Unit1.EventsData".TelemetryContent[11].KVP[37].Value)
   END_RUNG
   RUNG wire#w1
      Contact( true )
      { S7_Templates := "SrcType := LReal" } Mul(in1 := 0.0, in2 := 100.0, out => #data[37])
      { S7_Templates := "[SrcType := LReal, DestType := DInt]" } Convert(in := #data[37], out => "Unit1.EventsData".TelemetryContent[11].KVP[37].Value)
   END_RUNG
   // the same network as SCL:
   IF true AND false THEN "Unit1.EventsData".TelemetryContent[11].KVP[37].Value := 100; END_IF;
   IF true AND true THEN
       #data[37] := 0.0 * 100.0;
       "Unit1.EventsData".TelemetryContent[11].KVP[37].Value := LREAL_TO_DINT(#data[37]);
   END_IF;
END_REGION

REGION Network 39: PDR Data38
   RUNG wire#powerrail
      Contact( true )
      wire#w1
      Contact( false )
      Move(in := 100, out1 => "Unit1.EventsData".TelemetryContent[11].KVP[38].Value)
   END_RUNG
   RUNG wire#w1
      Contact( true )
      { S7_Templates := "SrcType := LReal" } Mul(in1 := 0.0, in2 := 100.0, out => #data[38])
      { S7_Templates := "[SrcType := LReal, DestType := DInt]" } Convert(in := #data[38], out => "Unit1.EventsData".TelemetryContent[11].KVP[38].Value)
   END_RUNG
   // the same network as SCL:
   IF true AND false THEN "Unit1.EventsData".TelemetryContent[11].KVP[38].Value := 100; END_IF;
   IF true AND true THEN
       #data[38] := 0.0 * 100.0;
       "Unit1.EventsData".TelemetryContent[11].KVP[38].Value := LREAL_TO_DINT(#data[38]);
   END_IF;
END_REGION

REGION Network 40: PDR Data39
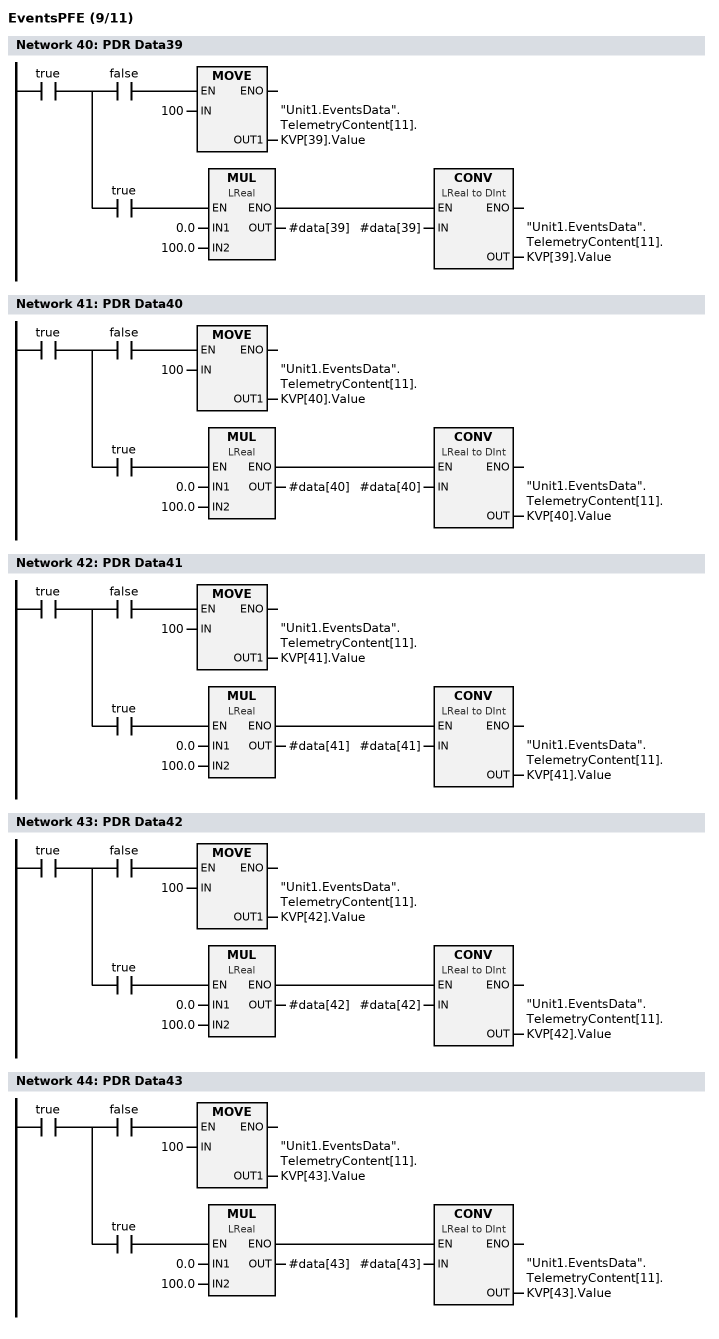
   RUNG wire#powerrail
      Contact( true )
      wire#w1
      Contact( false )
      Move(in := 100, out1 => "Unit1.EventsData".TelemetryContent[11].KVP[39].Value)
   END_RUNG
   RUNG wire#w1
      Contact( true )
      { S7_Templates := "SrcType := LReal" } Mul(in1 := 0.0, in2 := 100.0, out => #data[39])
      { S7_Templates := "[SrcType := LReal, DestType := DInt]" } Convert(in := #data[39], out => "Unit1.EventsData".TelemetryContent[11].KVP[39].Value)
   END_RUNG
   // the same network as SCL:
   IF true AND false THEN "Unit1.EventsData".TelemetryContent[11].KVP[39].Value := 100; END_IF;
   IF true AND true THEN
       #data[39] := 0.0 * 100.0;
       "Unit1.EventsData".TelemetryContent[11].KVP[39].Value := LREAL_TO_DINT(#data[39]);
   END_IF;
END_REGION

REGION Network 41: PDR Data40
   RUNG wire#powerrail
      Contact( true )
      wire#w1
      Contact( false )
      Move(in := 100, out1 => "Unit1.EventsData".TelemetryContent[11].KVP[40].Value)
   END_RUNG
   RUNG wire#w1
      Contact( true )
      { S7_Templates := "SrcType := LReal" } Mul(in1 := 0.0, in2 := 100.0, out => #data[40])
      { S7_Templates := "[SrcType := LReal, DestType := DInt]" } Convert(in := #data[40], out => "Unit1.EventsData".TelemetryContent[11].KVP[40].Value)
   END_RUNG
   // the same network as SCL:
   IF true AND false THEN "Unit1.EventsData".TelemetryContent[11].KVP[40].Value := 100; END_IF;
   IF true AND true THEN
       #data[40] := 0.0 * 100.0;
       "Unit1.EventsData".TelemetryContent[11].KVP[40].Value := LREAL_TO_DINT(#data[40]);
   END_IF;
END_REGION

REGION Network 42: PDR Data41
   RUNG wire#powerrail
      Contact( true )
      wire#w1
      Contact( false )
      Move(in := 100, out1 => "Unit1.EventsData".TelemetryContent[11].KVP[41].Value)
   END_RUNG
   RUNG wire#w1
      Contact( true )
      { S7_Templates := "SrcType := LReal" } Mul(in1 := 0.0, in2 := 100.0, out => #data[41])
      { S7_Templates := "[SrcType := LReal, DestType := DInt]" } Convert(in := #data[41], out => "Unit1.EventsData".TelemetryContent[11].KVP[41].Value)
   END_RUNG
   // the same network as SCL:
   IF true AND false THEN "Unit1.EventsData".TelemetryContent[11].KVP[41].Value := 100; END_IF;
   IF true AND true THEN
       #data[41] := 0.0 * 100.0;
       "Unit1.EventsData".TelemetryContent[11].KVP[41].Value := LREAL_TO_DINT(#data[41]);
   END_IF;
END_REGION

REGION Network 43: PDR Data42
   RUNG wire#powerrail
      Contact( true )
      wire#w1
      Contact( false )
      Move(in := 100, out1 => "Unit1.EventsData".TelemetryContent[11].KVP[42].Value)
   END_RUNG
   RUNG wire#w1
      Contact( true )
      { S7_Templates := "SrcType := LReal" } Mul(in1 := 0.0, in2 := 100.0, out => #data[42])
      { S7_Templates := "[SrcType := LReal, DestType := DInt]" } Convert(in := #data[42], out => "Unit1.EventsData".TelemetryContent[11].KVP[42].Value)
   END_RUNG
   // the same network as SCL:
   IF true AND false THEN "Unit1.EventsData".TelemetryContent[11].KVP[42].Value := 100; END_IF;
   IF true AND true THEN
       #data[42] := 0.0 * 100.0;
       "Unit1.EventsData".TelemetryContent[11].KVP[42].Value := LREAL_TO_DINT(#data[42]);
   END_IF;
END_REGION

REGION Network 44: PDR Data43
   RUNG wire#powerrail
      Contact( true )
      wire#w1
      Contact( false )
      Move(in := 100, out1 => "Unit1.EventsData".TelemetryContent[11].KVP[43].Value)
   END_RUNG
   RUNG wire#w1
      Contact( true )
      { S7_Templates := "SrcType := LReal" } Mul(in1 := 0.0, in2 := 100.0, out => #data[43])
      { S7_Templates := "[SrcType := LReal, DestType := DInt]" } Convert(in := #data[43], out => "Unit1.EventsData".TelemetryContent[11].KVP[43].Value)
   END_RUNG
   // the same network as SCL:
   IF true AND false THEN "Unit1.EventsData".TelemetryContent[11].KVP[43].Value := 100; END_IF;
   IF true AND true THEN
       #data[43] := 0.0 * 100.0;
       "Unit1.EventsData".TelemetryContent[11].KVP[43].Value := LREAL_TO_DINT(#data[43]);
   END_IF;
END_REGION

REGION Network 45: PDR Data44
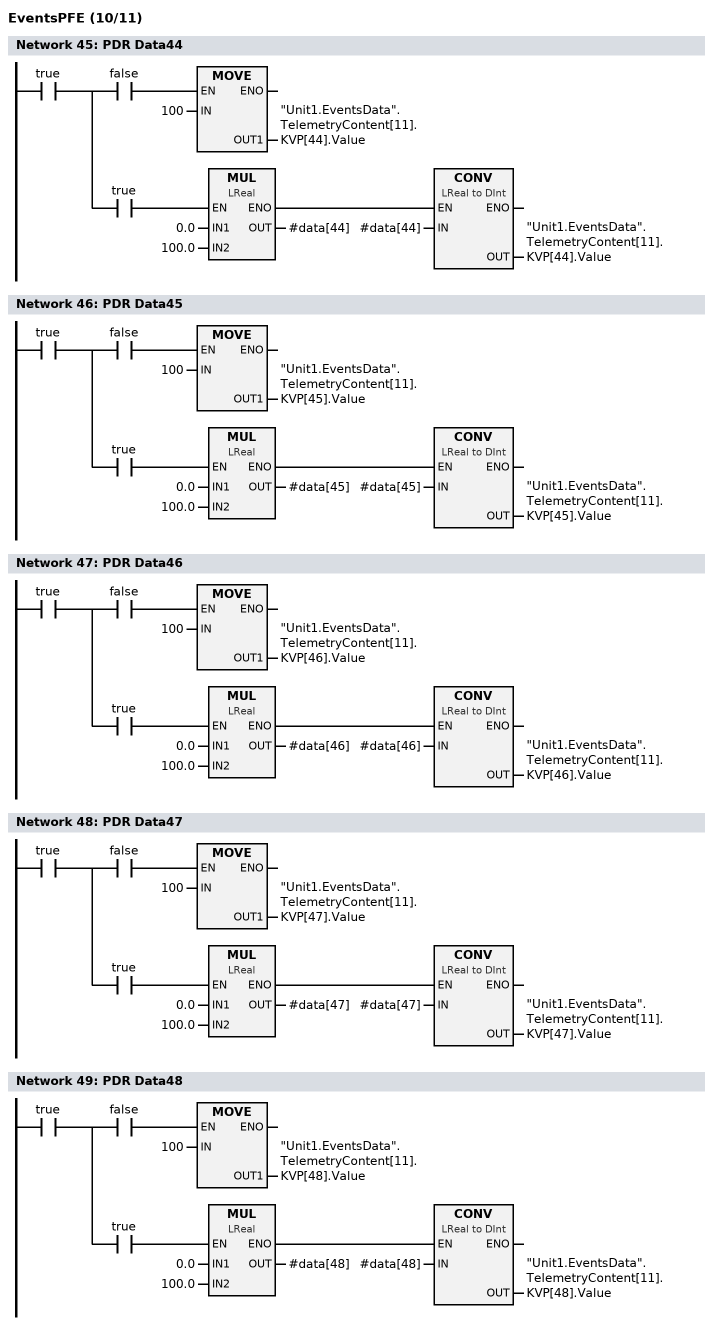
   RUNG wire#powerrail
      Contact( true )
      wire#w1
      Contact( false )
      Move(in := 100, out1 => "Unit1.EventsData".TelemetryContent[11].KVP[44].Value)
   END_RUNG
   RUNG wire#w1
      Contact( true )
      { S7_Templates := "SrcType := LReal" } Mul(in1 := 0.0, in2 := 100.0, out => #data[44])
      { S7_Templates := "[SrcType := LReal, DestType := DInt]" } Convert(in := #data[44], out => "Unit1.EventsData".TelemetryContent[11].KVP[44].Value)
   END_RUNG
   // the same network as SCL:
   IF true AND false THEN "Unit1.EventsData".TelemetryContent[11].KVP[44].Value := 100; END_IF;
   IF true AND true THEN
       #data[44] := 0.0 * 100.0;
       "Unit1.EventsData".TelemetryContent[11].KVP[44].Value := LREAL_TO_DINT(#data[44]);
   END_IF;
END_REGION

REGION Network 46: PDR Data45
   RUNG wire#powerrail
      Contact( true )
      wire#w1
      Contact( false )
      Move(in := 100, out1 => "Unit1.EventsData".TelemetryContent[11].KVP[45].Value)
   END_RUNG
   RUNG wire#w1
      Contact( true )
      { S7_Templates := "SrcType := LReal" } Mul(in1 := 0.0, in2 := 100.0, out => #data[45])
      { S7_Templates := "[SrcType := LReal, DestType := DInt]" } Convert(in := #data[45], out => "Unit1.EventsData".TelemetryContent[11].KVP[45].Value)
   END_RUNG
   // the same network as SCL:
   IF true AND false THEN "Unit1.EventsData".TelemetryContent[11].KVP[45].Value := 100; END_IF;
   IF true AND true THEN
       #data[45] := 0.0 * 100.0;
       "Unit1.EventsData".TelemetryContent[11].KVP[45].Value := LREAL_TO_DINT(#data[45]);
   END_IF;
END_REGION

REGION Network 47: PDR Data46
   RUNG wire#powerrail
      Contact( true )
      wire#w1
      Contact( false )
      Move(in := 100, out1 => "Unit1.EventsData".TelemetryContent[11].KVP[46].Value)
   END_RUNG
   RUNG wire#w1
      Contact( true )
      { S7_Templates := "SrcType := LReal" } Mul(in1 := 0.0, in2 := 100.0, out => #data[46])
      { S7_Templates := "[SrcType := LReal, DestType := DInt]" } Convert(in := #data[46], out => "Unit1.EventsData".TelemetryContent[11].KVP[46].Value)
   END_RUNG
   // the same network as SCL:
   IF true AND false THEN "Unit1.EventsData".TelemetryContent[11].KVP[46].Value := 100; END_IF;
   IF true AND true THEN
       #data[46] := 0.0 * 100.0;
       "Unit1.EventsData".TelemetryContent[11].KVP[46].Value := LREAL_TO_DINT(#data[46]);
   END_IF;
END_REGION

REGION Network 48: PDR Data47
   RUNG wire#powerrail
      Contact( true )
      wire#w1
      Contact( false )
      Move(in := 100, out1 => "Unit1.EventsData".TelemetryContent[11].KVP[47].Value)
   END_RUNG
   RUNG wire#w1
      Contact( true )
      { S7_Templates := "SrcType := LReal" } Mul(in1 := 0.0, in2 := 100.0, out => #data[47])
      { S7_Templates := "[SrcType := LReal, DestType := DInt]" } Convert(in := #data[47], out => "Unit1.EventsData".TelemetryContent[11].KVP[47].Value)
   END_RUNG
   // the same network as SCL:
   IF true AND false THEN "Unit1.EventsData".TelemetryContent[11].KVP[47].Value := 100; END_IF;
   IF true AND true THEN
       #data[47] := 0.0 * 100.0;
       "Unit1.EventsData".TelemetryContent[11].KVP[47].Value := LREAL_TO_DINT(#data[47]);
   END_IF;
END_REGION

REGION Network 49: PDR Data48
   RUNG wire#powerrail
      Contact( true )
      wire#w1
      Contact( false )
      Move(in := 100, out1 => "Unit1.EventsData".TelemetryContent[11].KVP[48].Value)
   END_RUNG
   RUNG wire#w1
      Contact( true )
      { S7_Templates := "SrcType := LReal" } Mul(in1 := 0.0, in2 := 100.0, out => #data[48])
      { S7_Templates := "[SrcType := LReal, DestType := DInt]" } Convert(in := #data[48], out => "Unit1.EventsData".TelemetryContent[11].KVP[48].Value)
   END_RUNG
   // the same network as SCL:
   IF true AND false THEN "Unit1.EventsData".TelemetryContent[11].KVP[48].Value := 100; END_IF;
   IF true AND true THEN
       #data[48] := 0.0 * 100.0;
       "Unit1.EventsData".TelemetryContent[11].KVP[48].Value := LREAL_TO_DINT(#data[48]);
   END_IF;
END_REGION

REGION Network 50: PDR Data49
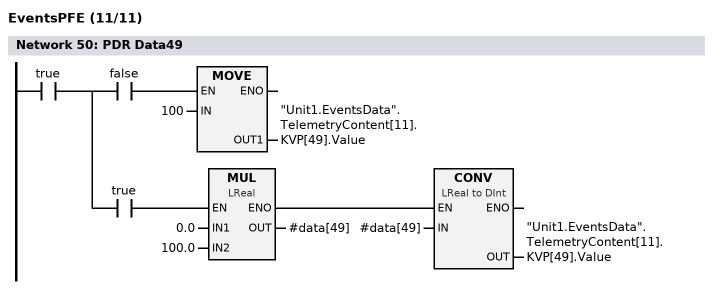
   RUNG wire#powerrail
      Contact( true )
      wire#w1
      Contact( false )
      Move(in := 100, out1 => "Unit1.EventsData".TelemetryContent[11].KVP[49].Value)
   END_RUNG
   RUNG wire#w1
      Contact( true )
      { S7_Templates := "SrcType := LReal" } Mul(in1 := 0.0, in2 := 100.0, out => #data[49])
      { S7_Templates := "[SrcType := LReal, DestType := DInt]" } Convert(in := #data[49], out => "Unit1.EventsData".TelemetryContent[11].KVP[49].Value)
   END_RUNG
   // the same network as SCL:
   IF true AND false THEN "Unit1.EventsData".TelemetryContent[11].KVP[49].Value := 100; END_IF;
   IF true AND true THEN
       #data[49] := 0.0 * 100.0;
       "Unit1.EventsData".TelemetryContent[11].KVP[49].Value := LREAL_TO_DINT(#data[49]);
   END_IF;
END_REGION
END_FUNCTION_BLOCK
